SYSTEM Performance
  (* Version 1.0, Author, Eclipse 4diac *)
  APPLICATION PerformanceApp
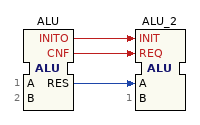
    FBS
      ALU : ALU(A := 1, B := 2);
      ALU_2 : ALU(B := 1);
    END_FBS
    EVENT_CONNECTIONS
      ALU.INITO TO ALU_2.INIT;
      ALU.CNF TO ALU_2.REQ;
    END_CONNECTIONS
    DATA_CONNECTIONS
      ALU.RES TO ALU_2.A;
    END_CONNECTIONS
  END_APPLICATION
END_SYSTEM
